{attribute 'qualified_only'}
{attribute 'strict'}
TYPE DUT :
(
	enum_member := 0
);
END_TYPE

(* stored: Version 1.1.0.1, ProductVersion 3.1.4024.15
   DUT DUT: Id {4d82e2ee-25cd-420c-ab73-fb322249dde6} *)
